(* IEC 61131-3 sources: stc/tests/opcua_golden/st301_shape, 6 files *)

(* ---- types.st ---- *)
TYPE E_DriveState :
(
	init := 0,
	cnf := 1,
	rdy := 2,
	run := 3
);
END_TYPE

TYPE E_402State :
(
	not_ready := 0,
	switch_on_disabled := 1,
	ready_to_switch_on := 2,
	fault := 3,
	switched_on := 4,
	operation_enabled := 5
);
END_TYPE

{attribute 'OPC.UA.DA.StructuredType' := '1'}
TYPE ST_Drive_HMI :
STRUCT
	p_cmd_JogFwd : BOOL;
	{attribute 'OPC.UA.DA.Access' := '1'}
	{attribute 'OPC.UA.DA.Description' := 'Drive fault'}
	p_stat_Error : BOOL;
	{attribute 'OPC.UA.DA.Access' := '1'}
	p_stat_State : E_DriveState;
	{attribute 'OPC.UA.DA.Access' := '1'}
	p_stat_402_State : E_402State;
	{attribute 'OPC.UA.DA.Access' := '1'}
	p_stat_Frequency : REAL;
	{attribute 'OPC.UA.DA.Access' := '1'}
	p_stat_SlaveId : UINT;
	p_cfg_AutoFreq : REAL;
END_STRUCT
END_TYPE

{attribute 'OPC.UA.DA.StructuredType' := '1'}
TYPE ST_Sensor_HMI :
STRUCT
	{attribute 'OPC.UA.DA.Access' := '1'}
	p_stat_xRaw : BOOL;
	p_cfg_Invert : BOOL;
END_STRUCT
END_TYPE

TYPE ST_Bus :
STRUCT
	nNodes : INT;
	xOk : BOOL;
END_STRUCT
END_TYPE

TYPE ST_ConveyorCfg :
STRUCT
	rMax : REAL;
	eMode : E_DriveState;
END_STRUCT
END_TYPE

(* ---- GVL_BatchLines.st ---- *)
VAR_GLOBAL
	Drives_Line1 : ARRAY[1..2] OF FB_Drive;
	{attribute 'OPC.UA.DA' := '2'}
	Internal_Bus_8 : ST_Bus;
	{attribute 'OPC.UA.DA' := '1'}
	{attribute 'OPC.UA.DA.Description' := 'Batches on line $'1$' ($$ counted)'}
	nBatchCount : DINT := 17;
	{attribute 'OPC.UA.DA' := '1'}
	Conveyor : FB_Conveyor;
END_VAR

(* ---- GVL_Roe.st ---- *)
VAR_GLOBAL
	{attribute 'OPC.UA.DA' := '1'}
	aRoe : ARRAY[0..3] OF INT := [1, 2, 3, 4];
END_VAR

(* ---- sensors.st ---- *)
VAR_GLOBAL
	EPW01_WA01_IS11 : FB_Sensor;
	EPW01_WA01_IS12 : FB_Sensor;
END_VAR

(* ---- fbs.st ---- *)
FUNCTION_BLOCK FB_Drive
VAR
	{attribute 'OPC.UA.DA' := '1'}
	HMI : ST_Drive_HMI;
	tmrStart : TON;
	pAxis : POINTER TO INT;
END_VAR
IF HMI.p_stat_State = E_DriveState.init THEN
	HMI.p_stat_State := E_DriveState.rdy;
	HMI.p_stat_402_State := E_402State.switched_on;
END_IF;
HMI.p_stat_Frequency := HMI.p_cfg_AutoFreq;
HMI.p_stat_Error := HMI.p_cmd_JogFwd AND HMI.p_cfg_AutoFreq < 0.0;
tmrStart(IN := HMI.p_cmd_JogFwd, PT := T#1S);
END_FUNCTION_BLOCK

FUNCTION_BLOCK FB_Sensor
VAR
	{attribute 'OPC.UA.DA' := '1'}
	HMI : ST_Sensor_HMI;
	xRawIn : BOOL;
END_VAR
HMI.p_stat_xRaw := xRawIn XOR HMI.p_cfg_Invert;
END_FUNCTION_BLOCK

FUNCTION_BLOCK FB_Conveyor
VAR
	xRun : BOOL;
	{attribute 'OPC.UA.DA' := '0'}
	tmrDelay : TON;
	pDrive : POINTER TO INT;
	{attribute 'OPC.UA.DA.Access' := '1'}
	rSpeed : REAL;
	Cfg : ST_ConveyorCfg;
END_VAR
tmrDelay(IN := xRun, PT := T#500MS);
IF tmrDelay.Q THEN
	rSpeed := Cfg.rMax;
ELSE
	rSpeed := 0.0;
END_IF;
END_FUNCTION_BLOCK

(* ---- main.st ---- *)
PROGRAM MAIN
VAR
	nCycle : DINT;
	xInit : BOOL;
	tmrCycle : TON;
END_VAR
xInit := TRUE;
nCycle := nCycle + 1;
tmrCycle(IN := xInit, PT := T#1S);
GVL_BatchLines.Drives_Line1[1]();
GVL_BatchLines.Drives_Line1[2]();
GVL_BatchLines.Conveyor();
sensors.EPW01_WA01_IS11();
sensors.EPW01_WA01_IS12();
END_PROGRAM
